PROGRAM MAIN
VAR
END_VAR


SFC_Test();

END_PROGRAM

(* stored: Version 1.1.0.1, ProductVersion 3.1.4022.10
   POU MAIN: Id {14a6314a-b8ec-4561-9e8e-6070d556fead}, SpecialFunc None *)
